TEXTLIST TextList_SubTank_circuit
  0 = 'circuit not filled'
  1 = 'white ink'
  2 = 'storage fluid'
   = ''
END_TEXTLIST

(* stored: Version 1.1.0.1, ProductVersion 3.1.4024.11
   TextList TextList_SubTank_circuit: Id {ce5e6a6e-373d-49f7-855a-f3253a9e751f} *)
